      L     "MAL1S019Par".Ilo.ILOMode;
      L     10;
      <>I   ;
      JC    I10;
// man on
      A     "MAL1S019Par".Ilo.GrCMDManOn[1];
      S     "G007G".Gr.InManual; // GENERAL ELEMENTS GERM 3
      S     "G145M".Gr.InManual; // Traveling  Drive Germatingbox 3
      S     "G149M".Gr.InManual; // Turning Screws Germinationbox 3
      S     "G144M".Gr.InManual; // Wall locking Germatingbox 3
      S     "G142M".Gr.InManual; // Backwall moving Germatingbox 3
      S     "G143M".Gr.InManual; // Discharger locking Germatingbox 3
      R     "MAL1S019Par".Ilo.GrCMDManOn[1];
// man off
      A     "MAL1S019Par".Ilo.GrCMDManOff[1];
      S     "G007G".Gr.CmdManualOff; // GENERAL ELEMENTS GERM 3
      R     "G007G".Gr.InManual; // GENERAL ELEMENTS GERM 3
      S     "G145M".Gr.CmdManualOff; // Traveling  Drive Germatingbox 3
      R     "G145M".Gr.InManual; // Traveling  Drive Germatingbox 3
      R     "G145M".USW14; // ILO-cmd
      R     "G145M".USW15; // ILO-cmd
      S     "G149M".Gr.CmdManualOff; // Turning Screws Germinationbox 3
      R     "G149M".Gr.InManual; // Turning Screws Germinationbox 3
      R     "G149M".USW14; // ILO-cmd
      R     "G149M".USW15; // ILO-cmd
      S     "G144M".Gr.CmdManualOff; // Wall locking Germatingbox 3
      R     "G144M".Gr.InManual; // Wall locking Germatingbox 3
      S     "G143M".Gr.CmdManualOff; // Discharger locking Germatingbox 3
      R     "G143M".Gr.InManual; // Discharger locking Germatingbox 3
      S     "G142M".Gr.CmdManualOff; // Backwall moving Germatingbox 3
      R     "G142M".Gr.InManual; // Backwall moving Germatingbox 3
      R     "MAL1S019Par".Ilo.GrCMDManOff[1];
      R     "MAL1S019Par".Ilo.GrCMDManAdditional.Cmd1[1];
      R     "MAL1S019Par".Ilo.GrCMDManAdditional.Cmd2[1];
// man start
      A     "G147M".A_2311_KCL01I1.InpTrue; // pushbutton "start screws"
      S     "G007G".Gr.CmdOn; // GENERAL ELEMENTS GERM 3
      S     "G007G".Gr.CmdContinue; // GENERAL ELEMENTS GERM 3
      S     "G149M".Gr.CmdOn; // Turning Screws Germinationbox 3
      S     "G149M".Gr.CmdContinue; // Turning Screws Germinationbox 3
      S     "G145M".Gr.CmdOn; // Traveling  Drive Germatingbox 3
      S     "G145M".Gr.CmdContinue; // Traveling  Drive Germatingbox 3
      A     "MAL1S019Par".Ilo.GrCMDManStart[1];
      R     "MAL1S019Par".Ilo.GrCMDManStart[1];
      A     "MAL1S019Par".Ilo.GrCMDManStart[2];
      R     "MAL1S019Par".Ilo.GrCMDManStart[2];
// man stop
      AN    "G147M".A_2311_KCL01I2.InpTrue; // pushbutton "stop screws"  //dyk 081025 Inverted
      S     "G149M".Gr.CmdOff; // Turning Screws Germinationbox 3
      A     "MAL1S019Par".Ilo.GrCMDManStop[1];
      O(    ;
      AN    "G147M".A_2311_KCL01I3.InpTrue; // pushbutton "drive fwd"
      AN    "G147M".A_2311_KCL01I4.InpTrue; // pushbutton "drive rev"
      )     ;
      S     "G145M".Gr.CmdOff; // Traveling  Drive Germatingbox 3

      AN    "G144M".Gr.InManual; // Wall locking Germatingbox 3
      O(    ;
      AN    "G147M".A_2315_KCL01I5.InpTrue; // pushbutton "locking"
      AN    "G147M".A_2315_KCL01I6.InpTrue; // pushbutton "unlocking"
      )     ;
      S     "G144M".Gr.CmdOff; // Wall locking/unlocking Germatingbox 3

      AN    "G143M".Gr.InManual; // discharger coupling Germatingbox 3
      O(    ;
      AN    "G147M".A_2315_KCL01I4.InpTrue; // pushbutton "discharger coupling"
      AN    "G147M".A_2315_KCL01I3.InpTrue; // pushbutton "discharger uncoupling"
      )     ;
      S     "G143M".Gr.CmdOff; // discharger coupling Germatingbox 3

      AN    "G142M".Gr.InManual; // Backwall moving Germatingbox 3
      O(    ;
      AN    "G147M".A_2315_KCL01I1.InpTrue; // pushbutton "backwall lifting"
      AN    "G147M".A_2315_KCL01I2.InpTrue; // pushbutton "backwall lowerring"
      )     ;
      S     "G142M".Gr.CmdOff; // Backwall moving Germatingbox 3

      A     "MAL1S019Par".Ilo.GrCMDManStop[1];
      R     "MAL1S019Par".Ilo.GrCMDManStop[1];
// man fault reset
      A     "MAL1S019Par".Ilo.GrCMDManFaultReset[1];
      S     "G007G".Gr.CmdFaultReset; // GENERAL ELEMENTS GERM 3
      S     "G145M".Gr.CmdFaultReset; // Traveling  Drive Germatingbox 3
      S     "G149M".Gr.CmdFaultReset; // Turning Screws Germinationbox 3
      R     "MAL1S019Par".Ilo.GrCMDManFaultReset[1];
      NOP   0;
// Manual wall locking
      AN    "G144M".Gr.InManual; // Wall locking Germatingbox 3
      ON    "G147M".A_2315_KCL01I5.InpTrue; // pushbutton "locking"
      JC    f102;
      S     "G144M".Gr.CmdOn; // Wall locking/unlocking Germatingbox 3
f102: NOP   0;
// Manual wall unlocking
      AN    "G144M".Gr.InManual; // Wall locking Germatingbox 3
      ON    "G147M".A_2315_KCL01I6.InpTrue; // pushbutton "unlocking"
      JC    f103;
      S     "G144M".Gr.CmdOn; // Wall locking/unlocking Germatingbox 3
f103: NOP   0;
// Manual discharger coupling
      AN    "G143M".Gr.InManual; // discharger coupling Germatingbox 3
      ON    "G147M".A_2315_KCL01I4.InpTrue; // pushbutton "discharger coupling"
      JC    f104;
      S     "G143M".Gr.CmdOn; // discharger coupling Germatingbox 3
f104: NOP   0;
// Manual discharger uncoupling
      AN    "G143M".Gr.InManual; // discharger coupling Germatingbox 3
      ON    "G147M".A_2315_KCL01I3.InpTrue; // pushbutton "discharger uncoupling"
      JC    f105;
      S     "G143M".Gr.CmdOn; // discharger coupling Germatingbox 3
f105: NOP   0;
// Manual backwall moving
      AN    "G142M".Gr.InManual; // Backwall moving Germatingbox 3
      ON    "G147M".A_2315_KCL01I1.InpTrue; // pushbutton "backwall lifting"
      JC    f106;
      S     "G142M".Gr.CmdOn; // Backwall moving Germatingbox 3
f106: NOP   0;
      AN    "G142M".Gr.InManual; // Backwall moving Germatingbox 3
      ON    "G147M".A_2315_KCL01I2.InpTrue; // pushbutton "backwall lowerring"
      JC    f107;
      S     "G142M".Gr.CmdOn; // Backwall moving Germatingbox 3
f107: NOP   0;
// manual direction
      AN    "G145M".Gr.InManual; // Traveling  Drive Germatingbox 3
      O     ;
      AN    "G147M".A_2311_KCL01I3.InpTrue; // pushbutton "drive fwd"
      AN    "G147M".A_2311_KCL01I4.InpTrue; // pushbutton "drive rev"
      JC    f109;
      A     "G147M".A_2311_KCL01I3.InpTrue; // pushbutton "drive fwd"
      =     "G145M".USW14; // ILO-cmd run fwd
      S     "G145M".Gr.CmdOn; // Traveling  Drive Germatingbox 3
      A     "G147M".A_2311_KCL01I4.InpTrue; // pushbutton "drive rev"
      =     "G145M".USW15; // ILO-cmd run rev
      S     "G145M".Gr.CmdOn; // Traveling  Drive Germatingbox 3

// target position
      L     "MAL1S019Par".Ilo.SetpointInt01[1];
      T     "MAL1S019Par".Par.ParIntProcess.Speed_ILO_FloorRotating;
f109: NOP   0;

I10:  NOP   0;
//
// copy state
      A     "G145M".Gr.InOutAutostartMan; // TRAVELLING DRIVE GERM 3
      =     "MAL1S019Par".Ilo.GrSTMan[2];
      A     "G149M".Gr.InOutAutostartMan; // TURNING SCREWS GERM 3
      =     "MAL1S019Par".Ilo.GrSTMan[6];
      A     "G150M".Gr.InOutAutostartMan; // FAN AND VALVE SRAY AIR GERM 3
      =     "MAL1S019Par".Ilo.GrSTMan[7];
      A     "G151M".Gr.InOutAutostartMan; // FRESH AIR LOUVER GERM 3
      =     "MAL1S019Par".Ilo.GrSTMan[8];
      A     "G157M".Gr.InOutAutostartMan; // COOLING / HEATING GERM 3
      =     "MAL1S019Par".Ilo.GrSTMan[14];

// copy state

NETWORK
TITLE =ASW_9999: Init ASW Flags
// clear all flags explicde to find them back
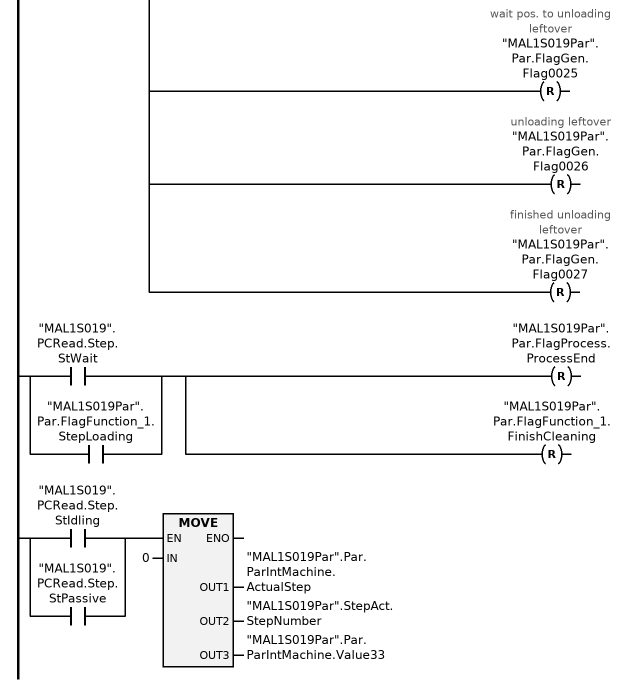
      A     "MAL1S019".PCRead.Step.StIdling;
      O     "MAL1S019".PCRead.Step.StPassive;
      R     "MAL1S019Par".Par.FlagFunction_1.StepLoading;
      R     "MAL1S019Par".Par.FlagFunction_1.StepUnloading;
      R     "MAL1S019Par".Par.FlagFunction_1.StepCleaning;
      R     "MAL1S019Par".Par.FlagFunction_1.LoadingBreak;
      R     "MAL1S019Par".Par.FlagFunction_1.UnloadingBreak;
      R     "MAL1S019Par".Par.FlagFunction_1.CleaningBreak;
      R     "MAL1S019Par".Par.FlagFunction_1.FinishLoading;
      R     "MAL1S019Par".Par.FlagFunction_1.FinishUnloading;
      R     "MAL1S019Par".Par.FlagFunction_1.FinishCleaning;
      R     "MAL1S019Par".Par.FlagFunction_1.Round_1;
      R     "MAL1S019Par".Par.FlagFunction_1.Round_2;
      R     "MAL1S019Par".Par.FlagFunction_1.Round_3;
      R     "MAL1S019Par".Par.FlagFunction_1.Round_4;
      R     "MAL1S019Par".Par.FlagFunction_1.Round_5;
      R     "MAL1S019Par".Par.FlagFunction_1.Round_6;
      R     "MAL1S019Par".Par.FlagFunction_1.Beladung_beendet;
      R     "MAL1S019Par".Par.FlagFunction_1.Entladerunden_erreicht;
      R     "MAL1S019Par".Par.FlagFunction_1.Reinigungsrunde_erreicht;
      R     "MAL1S019Par".Par.FlagGen.TurningStarted;
      R     "MAL1S019Par".Par.FlagFunction_1.TurningStart;
      R     "MAL1S019Par".Par.FlagFunction_1.TurningStop;
      R     "MAL1S019Par".Par.FlagFunction_1.TurningLeft;
      R     "MAL1S019Par".Par.FlagFunction_1.TurningRight;
      R     "MAL1S019Par".Par.FlagFunction_1.LoadFirstPartEnd;
      R     "MAL1S019Par".Par.FlagFunction_1.TurningWithSpraying;
      R     "MAL1S019Par".Par.FlagFunction_1.TurningWithoutSpraying;
      R     "MAL1S019Par".Par.FlagGen.TurningStarted;
      R     "MAL1S019Par".Par.FlagProcess2.Turning1WithoutSpraying;
      R     "MAL1S019Par".Par.FlagProcess2.Turning2WithoutSpraying;
      R     "MAL1S019Par".Par.FlagProcess2.Turning1WithSpraying;
      R     "MAL1S019Par".Par.FlagProcess2.Turning2WithSpraying;
      R     "MAL1S019Par".Par.FlagProcess2.Turning1WithDosing;
      R     "MAL1S019Par".Par.FlagProcess2.Turning2WithDosing;
      R     "MAL1S019Par".Par.FlagProcess2.StartFirstTurningRound;
      R     "MAL1S019Par".Par.FlagProcess2.StartSecondTurningRound;

      R     "MAL1S019Par".Par.FlagFunction_1.UnloadFirstPartEnd;
      R     "MAL1S019Par".Par.FlagFunction_1.UnloadSecondPartEnd;
      R     "MAL1S019Par".Par.FlagFunction_1.UnloadFirstPart;
      R     "MAL1S019Par".Par.FlagFunction_1.UnloadSecondPart;
      R     "MAL1S019Par".Par.FlagFunction_1.UnloadingStarted;
      R     "MAL1S019Par".Par.FlagProcess.ProcessActive;
      R     "MAL1S019Par".Par.FlagProcess.ProcessStartFP;
      R     "MAL1S019Par".Par.FlagProcess.ProcessStartScan;
      R     "MAL1S019Par".Par.FlagProcess.ProcessEnd;
      R     "MAL1S019Par".Par.FlagProcess.FP_SendResultToPIC;
      R     "MAL1S019Par".Par.FlagMachine.ImpulsNullstellung;
      R     "MAL1S019Par".Par.FlagMachine_0.CmdTurnRevAfterUnloading;
      R     "MAL1S019Par".Par.FlagMachine_0.CleaningAfterUnloading;
      R     "MAL1S019Par".Par.FlagMachine_0.CleaningAfterLoading;

      R     "MAL1S019Par".Par.FlagGen.Flag0024; // finished first unloading
      R     "MAL1S019Par".Par.FlagGen.Flag0025; // wait pos. to unloading leftover
      R     "MAL1S019Par".Par.FlagGen.Flag0026; // unloading leftover
      R     "MAL1S019Par".Par.FlagGen.Flag0027; // finished unloading leftover
//
      A     "MAL1S019".PCRead.Step.StWait;
      O     "MAL1S019Par".Par.FlagFunction_1.StepLoading;
      R     "MAL1S019Par".Par.FlagProcess.ProcessEnd;
      R     "MAL1S019Par".Par.FlagFunction_1.FinishCleaning;

      A     "MAL1S019".PCRead.Step.StIdling;
      O     "MAL1S019".PCRead.Step.StPassive;
      JCN   csn;
      L     0; // clear step number
      T     "MAL1S019Par".Par.ParIntMachine.ActualStep;
      T     "MAL1S019Par".StepAct.StepNumber;
      T     "MAL1S019Par".Par.ParIntMachine.Value33; //aktuelle Wartezeit Maschine bei 100% Unloading-Position
csn:  NOP   0;

NETWORK
TITLE =Main0_End: Init flag
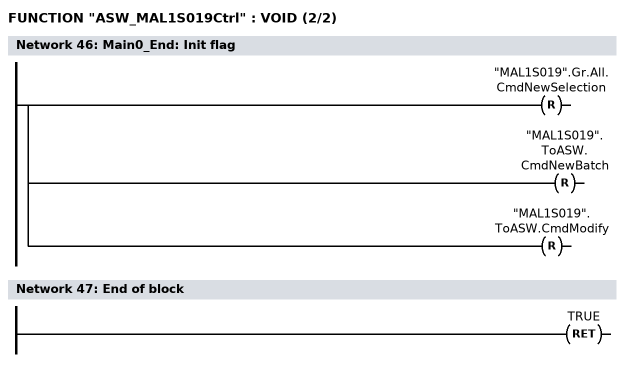

      SET   ;
      R     "MAL1S019".Gr.All.CmdNewSelection;
      R     "MAL1S019".ToASW.CmdNewBatch;
      R     "MAL1S019".ToASW.CmdModify;

NETWORK
TITLE =End of block

      BE    ;

END_FUNCTION

